PROGRAM CommitWith200SMART
VAR
END_VAR

END_PROGRAM

(* stored: Version 1.1.0.1, ProductVersion 3.1.4024.9
   POU CommitWith200SMART: Id {bbaeedba-2ab1-4d6f-8745-64e0b8ac1adb}, SpecialFunc None *)
